PROGRAM MAIN
VAR
END_VAR

END_PROGRAM

(* stored: Version 1.1.0.1
   POU MAIN: Id {59924d6e-8eaa-4217-b2ac-8b546949a560} *)
